TYPE TupleStruct_1:
    STRUCT
        field0: LREAL;
        field1: LREAL;
    END_STRUCT;
END_TYPE
